Yaskawa INFORM job: OK_R2_O55A(90,180)KMOK.JBI

/JOB
//NAME OK_R2_O55A(90,180)KMOK
//POS
///NPOS 386,386,386,17,0,0
///TOOL 0
///POSTYPE PULSE
///PULSE
C00000=-76403,1922,-14330,-35191,82947,48006
C00001=-78901,2717,-11338,-34802,80748,47687
C00002=-84368,8537,-7735,-27600,82156,45752
C00003=-85611,7008,-9073,-27350,81787,45371
C00004=-84730,8997,-7223,-27533,81967,45660
C00005=-84730,9088,-5441,-27593,81032,45882
C00006=-85090,9461,-6706,-27466,81778,45569
C00007=-85585,11950,-4488,-27371,81540,45439
C00008=-80569,4182,-8968,-34529,79490,47402
C00009=-79583,3757,-10261,-34677,80367,47529
C00010=-77101,2900,-13311,-35064,82560,47846
C00011=-78635,-10836,-23571,-6788,56023,46567
C00012=-80100,-6638,-17370,-6019,54259,46080
C00013=-81067,-4347,-13182,-5518,52796,45761
C00014=-81067,-4111,-11404,-5589,51829,45816
C00015=-81465,-3918,-12726,-5271,52710,45599
C00016=-81982,-3205,-12144,-4945,52685,45384
C00017=-81465,-3918,-12726,-5271,52710,45599
C00018=-79282,-7726,-17487,-6563,53838,46443
C00019=-77787,-11932,-23670,-7341,55599,46936
C00020=-71781,-30779,-36927,-16583,56350,53193
C00021=-76601,7892,12119,-36699,72044,51538
C00022=-79081,9717,16128,-36650,69746,51261
C00023=-82756,10272,16118,-32252,68446,49901
C00024=-83910,8771,14784,-32035,68048,49533
C00025=-82756,10272,16118,-32252,68446,49901
C00026=-82756,11092,18536,-32472,67538,50179
C00027=-82756,10272,16118,-32252,68446,49901
C00028=-83393,13264,18808,-32164,68102,49736
C00029=-82756,10272,16118,-32252,68446,49901
C00030=-79125,8186,14884,-36648,69710,51254
C00031=-76625,6364,10892,-36701,72010,51539
C00032=-78619,-8468,-7802,-7622,47602,47178
C00033=-80084,-3545,-911,-6819,45772,46643
C00034=-80849,-1134,3864,-6473,44020,46410
C00035=-80849,-591,5622,-6568,43222,46468
C00036=-80849,-1134,3864,-6473,44020,46410
C00037=-81794,988,5635,-5793,43949,45962
C00038=-80849,-1134,3864,-6473,44020,46410
C00039=-79264,-4301,-246,-7489,45053,47087
C00040=-77768,-9252,-7148,-8299,46887,47630
C00041=-73501,-22878,-17280,-17361,48294,53822
C00042=-76582,7918,12198,-36708,72023,51553
C00043=-79062,9745,16210,-36660,69725,51276
C00044=-85631,8937,11684,-26093,69417,48444
C00045=-86788,7574,10485,-25849,69089,48061
C00046=-85631,8937,11684,-26093,69417,48444
C00047=-85631,9727,14257,-26282,68355,48694
C00048=-85631,8937,11684,-26093,69417,48444
C00049=-86384,12817,15152,-25960,69054,48229
C00050=-80206,9359,17079,-36653,68644,51156
C00051=-79213,8529,15380,-36663,69568,51266
C00052=-76716,6688,11367,-36712,71869,51549
C00053=-78496,-8401,-7547,-7720,47491,47244
C00054=-79964,-3473,-648,-6917,45658,46708
C00055=-80829,339,5196,-6494,43959,46423
C00056=-80829,927,7090,-6597,43101,46485
C00057=-80829,339,5196,-6494,43959,46423
C00058=-81723,1584,6242,-5853,43887,45997
C00059=-80829,339,5196,-6494,43959,46423
C00060=-79396,-4326,-472,-7381,45166,47015
C00061=-77904,-9273,-7368,-8190,46997,47557
C00062=-73798,-22065,-16698,-17164,48289,53685
C00063=-76687,8147,12453,-36701,71947,51534
C00064=-79164,9987,16479,-36654,69648,51259
C00065=-85469,9101,11403,-25682,69642,48313
C00066=-87077,7212,9743,-25336,69193,47776
C00067=-85469,9101,11403,-25682,69642,48313
C00068=-85469,10017,14410,-25899,68394,48603
C00069=-85469,9101,11403,-25682,69642,48313
C00070=-86200,12844,14752,-25552,69292,48104
C00071=-80097,9169,16882,-36663,68709,51181
C00072=-79103,8344,15188,-36673,69634,51291
C00073=-76603,6515,11188,-36723,71934,51575
C00074=-78620,-8311,-7590,-7627,47551,47182
C00075=-80084,-3383,-689,-6825,45719,46647
C00076=-80782,-115,4996,-6540,43852,46454
C00077=-80782,405,6668,-6631,43097,46512
C00078=-80782,126,5782,-6582,43497,46482
C00079=-81646,1735,7133,-5954,43425,46068
C00080=-80263,-769,3748,-6862,44325,46668
C00081=-79285,-4364,-387,-7468,45105,47073
C00082=-77789,-9311,-7283,-8278,46937,47615
C00083=-72207,-27183,-21377,-18066,48871,54317
C00084=-76718,8235,12740,-36721,71828,51562
C00085=-79194,10089,16780,-36678,69527,51288
C00086=-85949,10651,13260,-25494,69998,48201
C00087=-87185,9191,11962,-25242,69663,47789
C00088=-85949,10651,13260,-25494,69998,48201
C00089=-85949,11213,15096,-25622,69235,48375
C00090=-85949,10898,14078,-25551,69656,48279
C00091=-86536,13982,16861,-25455,69360,48114
C00092=-80117,8915,16512,-36639,68779,51146
C00093=-79122,8093,14823,-36651,69703,51257
C00094=-76620,6271,10832,-36704,72003,51543
C00095=-78696,-8281,-7580,-7575,47554,47147
C00096=-80158,-3350,-677,-6772,45721,46612
C00097=-80887,125,5361,-6477,43742,46411
C00098=-80887,585,6834,-6555,43076,46460
C00099=-80887,270,5831,-6501,43529,46426
C00100=-81591,1736,7061,-5991,43471,46090
C00101=-79799,-2298,2499,-7195,44348,46889
C00102=-79220,-4347,-358,-7515,45102,47104
C00103=-77723,-9293,-7254,-8324,46936,47646
C00104=-72435,-26599,-20972,-17915,48869,54211
C00105=-76570,-17687,-14850,-19798,75838,26477
C00106=-76570,-17687,-14850,-19798,75838,26477
C00107=-87745,-9605,-5375,-17930,71662,23017
C00108=-89443,-6815,-2798,-17604,71148,22465
C00109=-89634,-5842,-2020,-17563,71128,22397
C00110=-89443,-6815,-2798,-17604,71148,22465
C00111=-89443,-7581,-5630,-17479,72437,22273
C00112=-91168,1721,1990,-17114,72156,21677
C00113=-91168,2041,3217,-17166,71590,21758
C00114=-91168,1721,1990,-17114,72156,21677
C00115=-82202,21106,36308,-50868,81053,24298
C00116=-83204,19644,34921,-50948,80572,24044
C00117=-78958,6455,21071,-50417,84024,24348
C00118=-86052,-24055,-21651,-18038,74505,23209
C00119=-69214,24096,20749,-23108,83460,36221
C00120=-71608,6597,4603,-68947,81663,-45930
C00121=-73755,7964,8737,-69115,79508,-45414
C00122=-74968,7560,10682,-69317,78154,-44963
C00123=-74968,8346,13234,-69526,77715,-44454
C00124=-74968,7560,10682,-69317,78154,-44963
C00125=-75623,8350,11378,-69309,77705,-45039
C00126=-73234,7979,11391,-69373,79243,-44640
C00127=-72371,7345,9649,-69271,80108,-44853
C00128=-70208,5990,5521,-69090,82272,-45369
C00129=-71458,6536,4837,-68973,81696,-45835
C00130=-73608,7910,8978,-69146,79540,-45319
C00131=-74773,7989,11985,-69422,78068,-44683
C00132=-74773,8525,13689,-69560,77778,-44345
C00133=-74773,8199,12662,-69476,77952,-44548
C00134=-75530,9339,13667,-69477,77429,-44630
C00135=-73160,8336,11414,-69348,79357,-44704
C00136=-72299,7709,9679,-69249,80221,-44917
C00137=-70142,6374,5567,-69075,82381,-45433
C00138=-71555,6569,4727,-68960,81663,-45884
C00139=-73704,8675,11428,-69316,79052,-44847
C00140=-74869,8697,12280,-69388,78072,-44775
C00141=-74869,9238,14009,-69531,77776,-44434
C00142=-74869,8887,12896,-69439,77966,-44653
C00143=-75513,9557,13488,-69438,77523,-44728
C00144=-73243,7935,11201,-69359,79273,-44682
C00145=-72380,7304,9463,-69258,80138,-44894
C00146=-70217,5958,5343,-69080,82301,-45410
C00147=-71620,7576,9372,-69242,80725,-44881
C00148=-73772,8435,11320,-69324,78986,-44831
C00149=-74875,8509,12078,-69384,78077,-44787
C00150=-74875,9056,13841,-69527,77773,-44437
C00151=-74875,8686,12655,-69431,77977,-44672
C00152=-75602,9232,13138,-69428,77479,-44758
C00153=-73284,7952,11199,-69357,79249,-44692
C00154=-72421,7320,9461,-69256,80114,-44904
C00155=-70258,5972,5339,-69078,82277,-45419
C00156=-71548,6406,4570,-68959,81673,-45889
C00157=-73698,8629,11672,-69344,78990,-44771
C00158=-74886,8172,11775,-69381,78074,-44795
C00159=-74886,8662,13358,-69511,77801,-44479
C00160=-74886,8307,12218,-69417,77997,-44706
C00161=-75624,9078,12897,-69416,77490,-44791
C00162=-73253,7959,11238,-69360,79262,-44679
C00163=-72390,7327,9499,-69259,80127,-44891
C00164=-70227,5979,5377,-69081,82290,-45407
C00165=-73684,21924,28477,-69535,76234,-41822
C00166=-74891,19654,26327,-69526,75480,-42047
C00167=-76506,21387,29456,-69805,74005,-41798
C00168=-74552,18110,24880,-69499,75745,-42046
C00169=-75381,18098,23573,-69331,75487,-42506
C00170=-77346,18837,26951,-69763,73526,-42008
C00171=-78427,17842,26055,-69366,71469,-52011
C00172=-78881,15304,23707,-69325,71217,-52134
C00173=-74815,19796,26463,-68977,79664,-56247
C00174=-73178,22919,29433,-68939,80676,-55936
C00175=-73666,19272,20464,-68833,77604,-43382
C00176=-74869,18380,22636,-69174,76106,-42756
C00177=-76554,20444,27119,-69566,74331,-42226
C00178=-74527,17435,22965,-69319,76074,-42409
C00179=-75357,17458,21697,-69150,75817,-42866
C00180=-76969,16913,23840,-69520,74127,-42370
C00181=-77511,13158,20364,-69473,73839,-42534
C00182=-77277,24403,30938,-69278,81382,-40713
C00183=-74792,18886,23871,-68814,80114,-56732
C00184=-73159,20683,22818,-68588,81821,-57193
C00185=-73710,21944,28497,-69536,76216,-41825
C00186=-74917,19676,26348,-69527,75461,-42050
C00187=-76528,21588,29866,-69843,73933,-41733
C00188=-74578,18131,24900,-69499,75726,-42049
C00189=-75407,18120,23593,-69332,75469,-42509
C00190=-76893,18416,26783,-69784,73785,-41898
C00191=-77360,15711,24383,-69770,73503,-41999
C00192=-77117,25124,33254,-69494,80031,-40440
C00193=-77229,28421,36396,-69270,82410,-39863
C00194=-74841,19817,26484,-68979,79646,-56250
C00195=-73204,22940,29453,-68940,80658,-55939
C00196=-73671,21913,28467,-69535,76243,-41821
C00197=-74878,19644,26317,-69525,75489,-42046
C00198=-76446,21696,29741,-69776,74042,-41781
C00199=-74539,18100,24870,-69498,75754,-42045
C00200=-75368,18087,23562,-69331,75496,-42505
C00201=-76829,18736,26940,-69733,73861,-41920
C00202=-77356,15298,23767,-69695,73575,-42071
C00203=-77179,22049,30100,-69528,78702,-40871
C00204=-77429,20567,28688,-69524,78574,-40949
C00205=-74802,19785,26453,-68977,79673,-56246
C00206=-73165,22909,29423,-68938,80686,-55935
C00207=-73697,21934,28487,-69536,76225,-41823
C00208=-74904,19665,26338,-69526,75471,-42049
C00209=-76487,21502,29779,-69838,73968,-41730
C00210=-74565,18121,24890,-69499,75735,-42048
C00211=-75394,18109,23583,-69331,75478,-42508
C00212=-76921,18139,26617,-69792,73759,-41884
C00213=-77416,14929,23641,-69755,73493,-42028
C00214=-76976,35689,43864,-68952,85010,-38929
C00215=-77187,33996,42040,-68958,84967,-39065
C00216=-74828,19807,26473,-68978,79655,-56248
C00217=-71271,31949,38327,-68936,81632,-55329
C00218=-64455,21408,16051,-68515,88030,-41500
C00219=-62220,-14655,-7588,-61843,66390,-57480
C00220=-65684,-34059,-16244,-44657,38104,-81353
C00221=-80507,10121,17600,-15341,57200,39800
C00222=-75845,16867,22558,-16973,58521,41505
C00223=-72897,41582,49979,-26317,62594,52964
C00224=-79860,8562,16225,-15575,57367,40041
C00225=-80508,9482,15745,-15208,57986,39686
C00226=-72982,41184,49489,-26278,62657,52914
C00227=-73697,37517,45702,-26032,62835,52576
C00228=-77058,24794,32654,-21193,59755,46647
C00229=-81408,13297,22074,-15190,55949,39611
C00230=-82232,11238,20195,-14857,55894,39277
C00231=-83257,9100,18238,-14442,55814,38864
C00232=-84450,6933,16333,-13966,55662,38392
C00233=-78697,11090,18471,-9995,55076,34572
C00234=-79295,11807,19109,-9744,54979,34335
C00235=-80544,10273,17728,-36477,70612,65921
C00236=-80540,10255,17715,-36477,70612,65923
C00237=-81663,12108,20960,-36551,69289,65897
C00238=-80539,9618,15857,-36320,71277,65692
C00239=-79786,11468,18802,-36578,70896,66153
C00240=-81901,13148,21842,-36522,69179,65831
C00241=-83549,20571,28688,-36398,68155,65466
C00242=-80537,10245,17705,-38455,66333,65488
C00243=-80540,10262,17718,-38454,66333,65487
C00244=-77732,-5014,-1669,-37983,70842,65115
C00245=-70423,-28857,-26484,-34936,42937,-87209
C00246=-72957,-20656,-20669,-25335,39181,70937
C00247=-76432,-9207,-9095,-22895,37031,69584
C00248=-77636,-3976,-2319,-22541,35326,69388
C00249=-76934,-7535,-7865,-22379,36987,69297
C00250=-76131,-8379,-7270,-23539,36472,69943
C00251=-76886,-1544,-324,-23246,35556,69779
C00252=-76079,1584,2343,-24028,35756,70214
C00253=-76929,-7527,-7764,-26477,38278,71586
C00254=-75666,-12476,-14553,-26648,40152,71669
C00255=-80539,4002,-16743,-13402,74658,37601
C00256=-80536,3873,-13936,-13516,72912,37797
C00257=-81546,5662,-9698,-13281,71105,37640
C00258=-79886,2359,-14058,-13789,72336,38095
C00259=-80534,3865,-14021,-13513,72959,37793
C00260=-82537,3680,-11348,-12920,70949,37307
C00261=-83585,1661,-13067,-12546,70807,36945
C00262=-84541,-32,-14546,-12201,70702,36611
C00263=-79182,4632,-13287,-8514,71050,33082
C00264=-78761,4323,-16471,-8590,72875,33101
C00265=-80569,4030,-12503,-34597,83280,61769
C00266=-80562,4114,-9678,-34698,81876,62211
C00267=-81659,4236,-6801,-34632,80014,62350
C00268=-80559,4091,-9841,-34693,81950,62189
C00269=-79806,5370,-7496,-34879,81603,62605
C00270=-82051,6116,-5182,-34562,79830,62247
C00271=-83492,12161,48,-34308,79156,61868
C00272=-83703,13184,961,-34271,79043,61817
C00273=-80556,4261,-7630,-36043,76415,61879
C00274=-80562,4081,-10441,-35844,77751,61431
C00275=-71462,-12551,-24032,-37751,81493,64028
C00276=-64215,-41183,-30200,-41548,42479,-83127
C00277=-75268,-8940,1587,-28059,31543,72401
C00278=-76569,-4731,4953,-26676,31199,71625
C00279=-77625,506,10820,-26265,30038,71368
C00280=-77071,-3623,4563,-25583,31771,71034
C00281=-76271,-4245,5350,-26977,31300,71794
C00282=-76971,2980,13032,-27029,30166,71792
C00283=-76158,6294,15992,-27966,30325,72317
C00284=-77064,-3050,6321,-30619,32600,73861
C00285=-75803,-7249,2926,-31827,33007,74555
C00286=-80516,10172,17645,-15338,57197,39797
C00287=-80517,10165,17644,-15338,57194,39797
C00288=-81429,13162,21998,-15186,55919,39607
C00289=-79869,8613,16269,-15572,57363,40038
C00290=-80517,9533,15790,-15205,57982,39683
C00291=-82245,11269,20291,-14856,55845,39281
C00292=-83580,8472,17804,-14322,55699,38749
C00293=-84398,6972,16513,-13999,55581,38427
C00294=-79088,10454,17905,-9826,55051,34413
C00295=-74888,4098,12338,-11562,55761,36069
C00296=-80552,10324,17774,-36476,70606,65919
C00297=-80549,10306,17761,-36476,70607,65921
C00298=-83683,7693,15438,-32682,67636,65344
C00299=-80548,9669,15902,-36319,71272,65690
C00300=-79795,11519,18847,-36577,70890,66151
C00301=-84004,9174,16701,-32630,67499,65250
C00302=-85602,16570,23210,-32388,66714,64811
C00303=-80546,10295,17751,-38454,66328,65486
C00304=-80549,10312,17763,-38453,66327,65485
C00305=-76939,-6698,-208,-38485,69790,65864
C00306=-67266,-29602,-13484,-36434,33447,77204
C00307=-75146,-9337,1276,-28189,31574,72475
C00308=-76453,-5135,4625,-26799,31231,71694
C00309=-77647,460,10904,-26298,29964,71381
C00310=-76958,-4030,4231,-25703,31802,71100
C00311=-76155,-4648,5022,-27099,31332,71863
C00312=-76931,2821,12923,-27078,30166,71815
C00313=-76073,5866,15538,-28006,30408,72336
C00314=-76950,-3457,5988,-30727,32638,73923
C00315=-75683,-7648,2608,-31942,33044,74622
C00316=-80508,8315,12089,-14954,59582,39461
C00317=-80505,9651,16284,-15248,57749,39721
C00318=-81490,12944,21701,-15149,55979,39575
C00319=-79855,8537,16203,-15577,57368,40043
C00320=-80504,9457,15722,-15209,57987,39688
C00321=-82467,11028,20074,-14770,55816,39193
C00322=-83319,9325,18634,-14437,55675,38860
C00323=-83964,7971,17403,-14174,55621,38599
C00324=-84422,7198,16724,-13991,55562,38417
C00325=-78819,10126,16706,-9875,55645,34468
C00326=-78596,10216,16456,-9945,55869,34539
C00327=-80539,10247,17706,-36477,70615,65922
C00328=-80536,10230,17693,-36477,70615,65924
C00329=-81604,11432,20382,-36558,69320,65911
C00330=-80534,9593,15834,-36320,71280,65693
C00331=-79781,11443,18779,-36578,70899,66154
C00332=-82039,13393,22124,-36517,69083,65803
C00333=-83392,19347,27632,-36414,68242,65504
C00334=-83616,20496,28669,-36395,68109,65452
C00335=-80533,10219,17683,-38456,66335,65489
C00336=-80536,10236,17695,-38455,66335,65488
C00337=-76398,-4716,5168,-39090,68227,66710
C00338=-67688,-28685,-12865,-36008,33343,76954
C00339=-75228,-9072,1484,-28102,31553,72426
C00340=-76531,-4865,4844,-26717,31210,71648
C00341=-77847,119,10662,-26106,29876,71275
C00342=-77033,-3758,4453,-25623,31782,71056
C00343=-76233,-4379,5241,-27017,31310,71817
C00344=-76936,2995,13152,-27116,30117,71837
C00345=-76130,6238,16052,-28051,30278,72358
C00346=-77026,-3185,6210,-30655,32612,73882
C00347=-75763,-7381,2820,-31865,33019,74577
C00348=-80512,10146,17623,-15339,57198,39799
C00349=-80513,10140,17621,-15339,57196,39799
C00350=-81500,13127,22067,-15170,55850,39589
C00351=-79864,8588,16247,-15574,57365,40040
C00352=-80513,9508,15768,-15206,57984,39684
C00353=-82364,10966,20070,-14819,55805,39239
C00354=-83277,9255,18611,-14462,55660,38880
C00355=-83996,7868,17423,-14178,55551,38597
C00356=-84389,7230,16943,-14028,55450,38448
C00357=-78699,12714,19934,-10002,55011,34578
C00358=-77475,15494,24062,-10661,54073,35179
C00359=-80548,10298,17751,-36476,70609,65920
C00360=-80545,10281,17738,-36477,70610,65922
C00361=-82679,9625,18013,-34629,68410,65635
C00362=-80543,9644,15879,-36319,71274,65691
C00363=-79790,11494,18824,-36577,70893,66152
C00364=-83022,11356,19462,-34579,68269,65534
C00365=-84222,16885,24482,-34449,67579,65242
C00366=-84495,18260,25693,-34414,67437,65171
C00367=-80541,10270,17728,-38455,66331,65487
C00368=-80544,10287,17740,-38454,66331,65486
C00369=-71600,-1949,10031,-39049,69350,68326
C00370=-71600,-1949,10031,-39049,69350,68326
C00371=-78766,16664,26924,-37375,68202,69313
C00372=-80481,18381,29464,-37332,66914,69021
C00373=-80571,20050,31036,-37349,66789,69027
C00374=-82589,28813,39248,-37227,65478,68604
C00375=-78367,25278,33930,-37393,68464,69394
C00376=-93563,26241,26451,4282,61542,63605
C00377=-96314,32508,36024,18641,58909,62055
C00378=-92113,24530,27996,5482,55270,70397
C00379=-92106,24462,27769,4672,55649,70406
C00380=-91576,23902,26334,-3618,58754,70962
C00381=-93650,12043,18084,-5384,52096,70498
C00382=-97507,8799,15190,-3438,51997,68869
C00383=-93212,4360,14554,-16260,47827,71925
C00384=-94425,-6257,-911,-4852,54321,70064
C00385=-44833,-55261,-28957,-41445,79036,76616
BC00000=349204,673109,1075175
BC00001=349204,673109,1075175
BC00002=349204,673109,1075175
BC00003=349204,673109,1075175
BC00004=349204,673109,1075175
BC00005=349204,673109,1075175
BC00006=349204,673109,1075175
BC00007=349204,673109,1075175
BC00008=349204,673109,1075175
BC00009=349204,673109,1075175
BC00010=349204,673109,1075175
BC00011=305088,674616,1075175
BC00012=305088,674616,1075175
BC00013=305088,674616,1075175
BC00014=305088,674616,1075175
BC00015=305088,674616,1075175
BC00016=305088,674616,1075175
BC00017=305088,674616,1075175
BC00018=305088,674616,1075175
BC00019=305088,674616,1075175
BC00020=314803,666681,1075175
BC00021=348681,674864,1042481
BC00022=348681,674864,1042481
BC00023=348681,674864,1042481
BC00024=348681,674864,1042481
BC00025=348681,674864,1042481
BC00026=348681,674864,1042481
BC00027=348681,674864,1042481
BC00028=348681,674864,1042481
BC00029=348681,674864,1042481
BC00030=348681,674864,1042481
BC00031=348681,674864,1042481
BC00032=304891,674718,1003525
BC00033=304891,674718,1003525
BC00034=304891,674718,1003525
BC00035=304891,674718,1003525
BC00036=304891,674718,1003525
BC00037=304891,674718,1003525
BC00038=304891,674718,1003525
BC00039=304891,674718,1003525
BC00040=304891,674718,1003525
BC00041=314838,666681,1004817
BC00042=348633,674683,878796
BC00043=348633,674683,878796
BC00044=348633,674683,878796
BC00045=348633,674683,878796
BC00046=348633,674683,878796
BC00047=348633,674683,878796
BC00048=348633,674683,878796
BC00049=348633,674683,878796
BC00050=348633,674683,878796
BC00051=348633,674683,878796
BC00052=348633,674683,878796
BC00053=305592,674868,842714
BC00054=305592,674868,842714
BC00055=305592,674868,842714
BC00056=305592,674868,842714
BC00057=305592,674868,842714
BC00058=305592,674868,842714
BC00059=305592,674868,842714
BC00060=305592,674868,842714
BC00061=305592,674868,842714
BC00062=314872,666681,843515
BC00063=348685,675197,716542
BC00064=348685,675197,716542
BC00065=348685,675197,716542
BC00066=348685,675197,716542
BC00067=348685,675197,716542
BC00068=348685,675197,716542
BC00069=348685,675197,716542
BC00070=348685,675197,716542
BC00071=348685,675197,716542
BC00072=348685,675197,716542
BC00073=348685,675197,716542
BC00074=305467,675287,679878
BC00075=305467,675287,679878
BC00076=305467,675287,679878
BC00077=305467,675287,679878
BC00078=305467,675287,679878
BC00079=305467,675287,679878
BC00080=305467,675287,679878
BC00081=305467,675287,679878
BC00082=305467,675287,679878
BC00083=314907,666681,682214
BC00084=348720,675488,554835
BC00085=348720,675488,554835
BC00086=348720,675488,554835
BC00087=348720,675488,554835
BC00088=348720,675488,554835
BC00089=348720,675488,554835
BC00090=348720,675488,554835
BC00091=348720,675488,554835
BC00092=348720,675488,554835
BC00093=348720,675488,554835
BC00094=348720,675488,554835
BC00095=305310,675530,518487
BC00096=305310,675530,518487
BC00097=305310,675530,518487
BC00098=305310,675530,518487
BC00099=305310,675530,518487
BC00100=305310,675530,518487
BC00101=305310,675530,518487
BC00102=305310,675530,518487
BC00103=305310,675530,518487
BC00104=314942,666681,520912
BC00105=378648,679076,578921
BC00106=378648,679076,319795
BC00107=378648,679076,319795
BC00108=378648,679076,319795
BC00109=378648,679076,319795
BC00110=378648,679076,319795
BC00111=378648,679076,319795
BC00112=378648,679076,319795
BC00113=378648,679076,319795
BC00114=378648,679076,319795
BC00115=378648,679076,319795
BC00116=378648,679076,319795
BC00117=378648,679076,319795
BC00118=378648,679076,319795
BC00119=378648,679076,578921
BC00120=398174,688559,405806
BC00121=398174,688559,405806
BC00122=398174,688559,405806
BC00123=398174,688559,405806
BC00124=398174,688559,405806
BC00125=398174,688559,405806
BC00126=398174,688559,405806
BC00127=398174,688559,405806
BC00128=398174,688559,405806
BC00129=398174,688393,568935
BC00130=398174,688393,568935
BC00131=398174,688393,568935
BC00132=398174,688393,568935
BC00133=398174,688393,568935
BC00134=398174,688393,568935
BC00135=398174,688393,568935
BC00136=398174,688393,568935
BC00137=398174,688393,568935
BC00138=398174,688149,730160
BC00139=398174,688149,730160
BC00140=398174,688149,730160
BC00141=398174,688149,730160
BC00142=398174,688149,730160
BC00143=398174,688149,730160
BC00144=398174,688149,730160
BC00145=398174,688149,730160
BC00146=398174,688149,730160
BC00147=398174,687828,892370
BC00148=398174,687828,892370
BC00149=398174,687828,892370
BC00150=398174,687828,892370
BC00151=398174,687828,892370
BC00152=398174,687828,892370
BC00153=398174,687828,892370
BC00154=398174,687828,892370
BC00155=398174,687828,892370
BC00156=398174,687735,1053470
BC00157=398174,687735,1053470
BC00158=398174,687735,1053470
BC00159=398174,687735,1053470
BC00160=398174,687735,1053470
BC00161=398174,687735,1053470
BC00162=398174,687735,1053470
BC00163=398174,687735,1053470
BC00164=398174,687735,1053470
BC00165=398174,675730,786203
BC00166=398174,679514,767318
BC00167=398174,681028,759764
BC00168=398174,681028,759764
BC00169=398174,681028,759764
BC00170=398174,679196,759749
BC00171=398174,676312,759427
BC00172=398174,676312,759427
BC00173=398174,682565,762575
BC00174=398174,680140,779769
BC00175=398174,675445,1075175
BC00176=398174,679229,1075175
BC00177=398174,680743,1075175
BC00178=398174,680743,1075175
BC00179=398174,680743,1075175
BC00180=398174,680743,1075175
BC00181=398174,680743,1075175
BC00182=398174,680743,1075175
BC00183=398174,682279,1075175
BC00184=398174,679854,1075175
BC00185=398174,676016,462794
BC00186=398174,679800,443908
BC00187=398174,681314,436354
BC00188=398174,681314,436354
BC00189=398174,681314,436354
BC00190=398174,681314,436354
BC00191=398174,681314,436354
BC00192=398174,681314,436354
BC00193=398174,681314,436354
BC00194=398174,682851,439165
BC00195=398174,680426,456359
BC00196=398174,675587,948311
BC00197=398174,679371,929426
BC00198=398174,680885,921868
BC00199=398174,680885,921872
BC00200=398174,680885,921872
BC00201=398174,680885,921868
BC00202=398174,680885,921868
BC00203=398174,680885,921868
BC00204=398174,680885,921868
BC00205=398174,682422,924682
BC00206=398174,679997,941876
BC00207=398174,675874,624095
BC00208=398174,679658,605210
BC00209=398174,681170,597651
BC00210=398174,681171,597656
BC00211=398174,681171,597656
BC00212=398174,681170,597651
BC00213=398174,681170,597651
BC00214=398174,681170,597651
BC00215=398174,681170,597651
BC00216=398174,682708,600466
BC00217=398174,680283,617660
BC00218=398174,666681,626567
BC00219=360198,666681,720930
BC00220=313360,666681,837312
BC00221=317534,668949,937568
BC00222=315368,674001,918688
BC00223=314501,676022,911136
BC00224=314501,676022,911136
BC00225=314501,676022,911136
BC00226=314501,676022,911136
BC00227=314501,676022,911136
BC00228=314501,676022,911136
BC00229=314501,676022,911136
BC00230=314501,676022,911136
BC00231=314501,676022,911136
BC00232=314501,676022,911136
BC00233=293205,672518,918719
BC00234=294306,667154,937598
BC00235=358411,669398,910199
BC00236=352988,671786,892375
BC00237=350819,672740,885243
BC00238=350819,672741,885245
BC00239=350819,672741,885245
BC00240=350819,672741,885245
BC00241=350819,672741,885245
BC00242=349387,669987,879930
BC00243=354654,666972,897113
BC00244=354755,666681,897949
BC00245=313290,666681,1075175
BC00246=299789,666220,1075175
BC00247=298966,666220,1075175
BC00248=298637,666220,1075175
BC00249=298637,666220,1075175
BC00250=298637,666220,1075175
BC00251=298637,666220,1075175
BC00252=298637,666220,1075175
BC00253=311807,666220,1075175
BC00254=312962,666220,1075175
BC00255=317588,668663,1075175
BC00256=315422,673716,1075175
BC00257=314555,675737,1075175
BC00258=314555,675737,1075175
BC00259=314555,675737,1075175
BC00260=314556,675736,1075175
BC00261=314556,675736,1075175
BC00262=314556,675736,1075175
BC00263=293260,672232,1075175
BC00264=294360,666869,1075175
BC00265=358465,669112,1075175
BC00266=353042,671500,1075175
BC00267=350873,672456,1075175
BC00268=350873,672456,1075175
BC00269=350873,672456,1075175
BC00270=350873,672456,1075175
BC00271=350873,672456,1075175
BC00272=350873,672456,1075175
BC00273=349450,669548,1075175
BC00274=354717,666534,1075175
BC00275=354685,666681,1075175
BC00276=313430,666681,513902
BC00277=299680,666220,513222
BC00278=298858,666220,494557
BC00279=298529,666220,487091
BC00280=298529,666220,487091
BC00281=298529,666220,487091
BC00282=298529,666220,487091
BC00283=298529,666220,487091
BC00284=311698,666220,494536
BC00285=312853,666220,513199
BC00286=317480,669234,614158
BC00287=315313,674287,595278
BC00288=314447,676308,587726
BC00289=314447,676308,587726
BC00290=314447,676308,587726
BC00291=314447,676308,587726
BC00292=314447,676308,587726
BC00293=314447,676308,587726
BC00294=293151,672804,595309
BC00295=294252,667440,614188
BC00296=358357,669683,586789
BC00297=352934,672071,568965
BC00298=350764,673027,561835
BC00299=350764,673027,561835
BC00300=350764,673027,561835
BC00301=350764,673027,561835
BC00302=350764,673027,561835
BC00303=349300,670887,556521
BC00304=354567,667872,573704
BC00305=354825,666681,574539
BC00306=299762,666220,998740
BC00307=299762,666220,998740
BC00308=298939,666220,980075
BC00309=298610,666220,972608
BC00310=298610,666220,972608
BC00311=298610,666220,972608
BC00312=298610,666220,972608
BC00313=298610,666220,972608
BC00314=311779,666220,980053
BC00315=312935,666220,998717
BC00316=317561,668805,1075175
BC00317=315395,673858,1075175
BC00318=314528,675879,1073244
BC00319=314528,675879,1073244
BC00320=314528,675879,1073244
BC00321=314528,675879,1073244
BC00322=314528,675879,1073244
BC00323=314528,675879,1073244
BC00324=314528,675879,1073244
BC00325=293232,672375,1075175
BC00326=294333,667011,1075175
BC00327=358439,669255,1072306
BC00328=353015,671643,1054482
BC00329=350846,672598,1047353
BC00330=350846,672598,1047353
BC00331=350846,672598,1047353
BC00332=350846,672598,1047353
BC00333=350846,672598,1047353
BC00334=350846,672598,1047353
BC00335=349348,671076,1042041
BC00336=354615,668061,1059224
BC00337=354720,666681,1060057
BC00338=299707,666220,674523
BC00339=299707,666220,674523
BC00340=298885,666220,655858
BC00341=298556,666220,648392
BC00342=298556,666220,648392
BC00343=298556,666220,648392
BC00344=298556,666220,648392
BC00345=298556,666220,648392
BC00346=311725,666220,655837
BC00347=312880,666220,674501
BC00348=317507,669092,775460
BC00349=315340,674145,756580
BC00350=314474,676166,749028
BC00351=314474,676166,749028
BC00352=314474,676166,749028
BC00353=314474,676166,749028
BC00354=314474,676166,749028
BC00355=314474,676166,749028
BC00356=314474,676166,749028
BC00357=293178,672661,756610
BC00358=294279,667297,775489
BC00359=358384,669541,748090
BC00360=352961,671929,730266
BC00361=350791,672884,723137
BC00362=350791,672884,723137
BC00363=350791,672884,723137
BC00364=350791,672884,723137
BC00365=350791,672884,723137
BC00366=350791,672884,723137
BC00367=349368,669977,717821
BC00368=354635,666962,735004
BC00369=354635,666962,735004
BC00370=343366,666962,351655
BC00371=343366,666962,351655
BC00372=343366,666962,351655
BC00373=343366,666962,351655
BC00374=343366,666962,351655
BC00375=343366,666962,351655
BC00376=343366,666962,351655
BC00377=343366,666962,351655
BC00378=343366,666962,351655
BC00379=343366,666962,351655
BC00380=343366,666962,351655
BC00381=343366,666962,351655
BC00382=343366,666962,351655
BC00383=343366,666962,351655
BC00384=343366,666962,351655
BC00385=354635,666962,735004
EC00000=798156,1112951
EC00001=798156,1112951
EC00002=798156,1112951
EC00003=798156,1112951
EC00004=798156,1112951
EC00005=798156,1112951
EC00006=798156,1112951
EC00007=798156,1112951
EC00008=798156,1112951
EC00009=798156,1112951
EC00010=798156,1112951
EC00011=798156,1112951
EC00012=798156,1112951
EC00013=798156,1112951
EC00014=798156,1112951
EC00015=798156,1112951
EC00016=798156,1112951
EC00017=798156,1112951
EC00018=798156,1112951
EC00019=798156,1112951
EC00020=798156,1112951
EC00021=798156,1112951
EC00022=798156,1112951
EC00023=798156,1112951
EC00024=798156,1112951
EC00025=798156,1112951
EC00026=798156,1112951
EC00027=798156,1112951
EC00028=798156,1112951
EC00029=798156,1112951
EC00030=798156,1112951
EC00031=798156,1112951
EC00032=798156,1112951
EC00033=798156,1112951
EC00034=798156,1112951
EC00035=798156,1112951
EC00036=798156,1112951
EC00037=798156,1112951
EC00038=798156,1112951
EC00039=798156,1112951
EC00040=798156,1112951
EC00041=798156,1112951
EC00042=798156,1112951
EC00043=798156,1112951
EC00044=798156,1112951
EC00045=798156,1112951
EC00046=798156,1112951
EC00047=798156,1112951
EC00048=798156,1112951
EC00049=798156,1112951
EC00050=798156,1112951
EC00051=798156,1112951
EC00052=798156,1112951
EC00053=798156,1112951
EC00054=798156,1112951
EC00055=798156,1112951
EC00056=798156,1112951
EC00057=798156,1112951
EC00058=798156,1112951
EC00059=798156,1112951
EC00060=798156,1112951
EC00061=798156,1112951
EC00062=798156,1112951
EC00063=798156,1112951
EC00064=798156,1112951
EC00065=798156,1112951
EC00066=798156,1112951
EC00067=798156,1112951
EC00068=798156,1112951
EC00069=798156,1112951
EC00070=798156,1112951
EC00071=798156,1112951
EC00072=798156,1112951
EC00073=798156,1112951
EC00074=798156,1112951
EC00075=798156,1112951
EC00076=798156,1112951
EC00077=798156,1112951
EC00078=798156,1112951
EC00079=798156,1112951
EC00080=798156,1112951
EC00081=798156,1112951
EC00082=798156,1112951
EC00083=798156,1112951
EC00084=798156,1112951
EC00085=798156,1112951
EC00086=798156,1112951
EC00087=798156,1112951
EC00088=798156,1112951
EC00089=798156,1112951
EC00090=798156,1112951
EC00091=798156,1112951
EC00092=798156,1112951
EC00093=798156,1112951
EC00094=798156,1112951
EC00095=798156,1112951
EC00096=798156,1112951
EC00097=798156,1112951
EC00098=798156,1112951
EC00099=798156,1112951
EC00100=798156,1112951
EC00101=798156,1112951
EC00102=798156,1112951
EC00103=798156,1112951
EC00104=798156,1112951
EC00105=798156,1112951
EC00106=798156,1112951
EC00107=798156,1112951
EC00108=798156,1112951
EC00109=798156,1112951
EC00110=798156,1112951
EC00111=798156,1112951
EC00112=798156,1112951
EC00113=798156,1112951
EC00114=798156,1112951
EC00115=798156,1112951
EC00116=798156,1112951
EC00117=798156,1112951
EC00118=798156,1112951
EC00119=798156,1112951
EC00120=798156,1112951
EC00121=798156,1112951
EC00122=798156,1112951
EC00123=798156,1112951
EC00124=798156,1112951
EC00125=798156,1112951
EC00126=798156,1112951
EC00127=798156,1112951
EC00128=798156,1112951
EC00129=798156,1112951
EC00130=798156,1112951
EC00131=798156,1112951
EC00132=798156,1112951
EC00133=798156,1112951
EC00134=798156,1112951
EC00135=798156,1112951
EC00136=798156,1112951
EC00137=798156,1112951
EC00138=798156,1112951
EC00139=798156,1112951
EC00140=798156,1112951
EC00141=798156,1112951
EC00142=798156,1112951
EC00143=798156,1112951
EC00144=798156,1112951
EC00145=798156,1112951
EC00146=798156,1112951
EC00147=798156,1112951
EC00148=798156,1112951
EC00149=798156,1112951
EC00150=798156,1112951
EC00151=798156,1112951
EC00152=798156,1112951
EC00153=798156,1112951
EC00154=798156,1112951
EC00155=798156,1112951
EC00156=798156,1112951
EC00157=798156,1112951
EC00158=798156,1112951
EC00159=798156,1112951
EC00160=798156,1112951
EC00161=798156,1112951
EC00162=798156,1112951
EC00163=798156,1112951
EC00164=798156,1112951
EC00165=798156,1112951
EC00166=798156,1112951
EC00167=798156,1112951
EC00168=798156,1112951
EC00169=798156,1112951
EC00170=798156,1112951
EC00171=798156,1112951
EC00172=798156,1112951
EC00173=798156,1112951
EC00174=798156,1112951
EC00175=798156,1112951
EC00176=798156,1112951
EC00177=798156,1112951
EC00178=798156,1112951
EC00179=798156,1112951
EC00180=798156,1112951
EC00181=798156,1112951
EC00182=798156,1112951
EC00183=798156,1112951
EC00184=798156,1112951
EC00185=798156,1112951
EC00186=798156,1112951
EC00187=798156,1112951
EC00188=798156,1112951
EC00189=798156,1112951
EC00190=798156,1112951
EC00191=798156,1112951
EC00192=798156,1112951
EC00193=798156,1112951
EC00194=798156,1112951
EC00195=798156,1112951
EC00196=798156,1112951
EC00197=798156,1112951
EC00198=798152,1112950
EC00199=798156,1112951
EC00200=798156,1112951
EC00201=798152,1112950
EC00202=798152,1112950
EC00203=798152,1112950
EC00204=798152,1112950
EC00205=798156,1112951
EC00206=798156,1112951
EC00207=798156,1112951
EC00208=798156,1112951
EC00209=798153,1112948
EC00210=798156,1112951
EC00211=798156,1112951
EC00212=798153,1112948
EC00213=798153,1112948
EC00214=798153,1112948
EC00215=798153,1112948
EC00216=798156,1112951
EC00217=798156,1112951
EC00218=798156,1112951
EC00219=798156,1112951
EC00220=798156,1112951
EC00221=798156,1112951
EC00222=798156,1112951
EC00223=798156,1112951
EC00224=798156,1112951
EC00225=798156,1112951
EC00226=798156,1112951
EC00227=798156,1112951
EC00228=798156,1112951
EC00229=798156,1112951
EC00230=798156,1112951
EC00231=798156,1112951
EC00232=798156,1112951
EC00233=798156,1112951
EC00234=798156,1112951
EC00235=798156,1112951
EC00236=798156,1112951
EC00237=798154,1112950
EC00238=798156,1112951
EC00239=798156,1112951
EC00240=798156,1112951
EC00241=798156,1112951
EC00242=798156,1112951
EC00243=798156,1112951
EC00244=798156,1112951
EC00245=798156,1112951
EC00246=798156,1112951
EC00247=798156,1112951
EC00248=798156,1112951
EC00249=798156,1112951
EC00250=798156,1112951
EC00251=798156,1112951
EC00252=798156,1112951
EC00253=798156,1112951
EC00254=798156,1112951
EC00255=798156,1112951
EC00256=798156,1112951
EC00257=798156,1112951
EC00258=798156,1112951
EC00259=798156,1112951
EC00260=798155,1112950
EC00261=798155,1112950
EC00262=798155,1112950
EC00263=798156,1112951
EC00264=798156,1112951
EC00265=798156,1112951
EC00266=798156,1112951
EC00267=798156,1112951
EC00268=798156,1112951
EC00269=798156,1112951
EC00270=798156,1112951
EC00271=798156,1112951
EC00272=798156,1112951
EC00273=798156,1112951
EC00274=798156,1112951
EC00275=798156,1112951
EC00276=798156,1112951
EC00277=798156,1112951
EC00278=798156,1112951
EC00279=798156,1112951
EC00280=798156,1112951
EC00281=798156,1112951
EC00282=798156,1112951
EC00283=798156,1112951
EC00284=798156,1112951
EC00285=798156,1112951
EC00286=798156,1112951
EC00287=798156,1112951
EC00288=798156,1112951
EC00289=798156,1112951
EC00290=798156,1112951
EC00291=798156,1112951
EC00292=798156,1112951
EC00293=798156,1112951
EC00294=798156,1112951
EC00295=798156,1112951
EC00296=798156,1112951
EC00297=798156,1112951
EC00298=798156,1112951
EC00299=798156,1112951
EC00300=798156,1112951
EC00301=798156,1112951
EC00302=798156,1112951
EC00303=798156,1112951
EC00304=798156,1112951
EC00305=798156,1112951
EC00306=798156,1112951
EC00307=798156,1112951
EC00308=798156,1112951
EC00309=798156,1112951
EC00310=798156,1112951
EC00311=798156,1112951
EC00312=798156,1112951
EC00313=798156,1112951
EC00314=798156,1112951
EC00315=798156,1112951
EC00316=798156,1112951
EC00317=798156,1112951
EC00318=798156,1112951
EC00319=798156,1112951
EC00320=798156,1112951
EC00321=798156,1112951
EC00322=798156,1112951
EC00323=798156,1112951
EC00324=798156,1112951
EC00325=798156,1112951
EC00326=798156,1112951
EC00327=798156,1112951
EC00328=798156,1112951
EC00329=798156,1112951
EC00330=798156,1112951
EC00331=798156,1112951
EC00332=798156,1112951
EC00333=798156,1112951
EC00334=798156,1112951
EC00335=798156,1112951
EC00336=798156,1112951
EC00337=798156,1112951
EC00338=798156,1112951
EC00339=798156,1112951
EC00340=798156,1112951
EC00341=798156,1112951
EC00342=798156,1112951
EC00343=798156,1112951
EC00344=798156,1112951
EC00345=798156,1112951
EC00346=798156,1112951
EC00347=798156,1112951
EC00348=798156,1112951
EC00349=798156,1112951
EC00350=798156,1112951
EC00351=798156,1112951
EC00352=798156,1112951
EC00353=798156,1112951
EC00354=798156,1112951
EC00355=798156,1112951
EC00356=798156,1112951
EC00357=798156,1112951
EC00358=798156,1112951
EC00359=798156,1112951
EC00360=798156,1112951
EC00361=798156,1112951
EC00362=798156,1112951
EC00363=798156,1112951
EC00364=798156,1112951
EC00365=798156,1112951
EC00366=798156,1112951
EC00367=798156,1112951
EC00368=798156,1112951
EC00369=798156,1112951
EC00370=798156,1112951
EC00371=798156,1112951
EC00372=798156,1112951
EC00373=798156,1112951
EC00374=798156,1112951
EC00375=798156,1112951
EC00376=798156,1112951
EC00377=798156,1112951
EC00378=798156,1112951
EC00379=798156,1112951
EC00380=798156,1112951
EC00381=798156,1112951
EC00382=798156,1112951
EC00383=798156,1112951
EC00384=798156,1112951
EC00385=798156,1112951
///POSTYPE BASE
///RECTAN
///RCONF 0,0,0,0,0,0,0,0,0,0,0,0,0,0,0,0,0,0,0,0,0,0,0,0
P00006=0.222,-3.123,-1.508,0.0000,0.0000,0.0000
P00021=-0.225,-6.128,-0.405,0.0000,0.0000,0.0000
P00022=0.222,-3.123,-1.508,0.0000,0.0000,0.0000
P00023=0.143,-0.036,0.682,0.0000,0.0000,0.0000
P00031=1.853,-0.001,-1.549,0.0000,0.0000,0.0000
P00032=1.957,0.503,-7.217,0.0000,0.0000,0.0000
///RCONF 0,0,0,0,1,0,0,0,0,0,0,0,0,0,0,0,0,0,0,0,0,0,0,0
P00033=-0.123,0.612,-5.012,0.0000,0.0000,0.0000
///RCONF 0,0,0,0,0,0,0,0,0,0,0,0,0,0,0,0,0,0,0,0,0,0,0,0
P00041=0.192,3.924,0.305,0.0000,0.0000,0.0000
P00042=-0.217,1.941,0.413,0.0000,0.0000,0.0000
P00043=-0.044,-1.937,1.197,0.0000,0.0000,0.0000
P00051=0.367,3.892,0.009,0.0000,0.0000,0.0000
P00052=0.088,2.832,-0.342,0.0000,0.0000,0.0000
P00053=0.134,6.594,0.107,0.0000,0.0000,0.0000
P00061=1.575,-3.405,-0.752,0.0000,0.0000,0.0000
P00062=-0.135,-0.848,-1.706,0.0000,0.0000,0.0000
P00063=0.036,-0.654,-3.005,0.0000,0.0000,0.0000
P00100=1.890,0.539,-2.641,0.0000,0.0000,0.0000
//INST
///DATE 2025/02/07 18:49
///ATTR SC,RW
///GROUP1 RB1,BS1
///GROUP2 ST1
NOP
'MUZYLO 300124
'MUZYLO 310124
'POPRAWA I SPAWANIE
'OK_R2_o55a(90,180)
'Path S3739
SFTOF3D
CALL JOB:CLEAN-R1_KM_NEW
MOVJ C00000 BC00000 VJ=100.00  +MOVJ EC00000 VJ=100.00
MOVL C00001 BC00001 V=133.3  +MOVJ EC00001 VJ=100.00
SMOVL C00002 BC00002 V=83.3  +MOVJ EC00002
SREFP 3 C00003 BC00003  +REFP EC00003
CALL JOB:SEARCH-R1-S13D
SET P021 P006
SFTON3D P021
SMOVL C00004 BC00004 V=83.3  +MOVJ EC00004
SREFP 3 C00005 BC00005  +REFP EC00005
CALL JOB:SEARCH-R1-S13D
SET P021 P006
SFTON3D P021
SMOVL C00006 BC00006 V=83.3  +MOVJ EC00006
SREFP 3 C00007 BC00007  +REFP EC00007
CALL JOB:SEARCH-R1-S13D
SET P021 P006
SFTON3D P021
SMOVL C00008 BC00008 V=83.3  +MOVJ EC00008
MOVL C00009 BC00009 V=166.7  +MOVJ EC00009 VJ=100.00
MOVL C00010 BC00010 V=250.0  +MOVJ EC00010 VJ=100.00
'Path S3740
SFTOF3D
MOVJ C00011 BC00011 VJ=100.00  +MOVJ EC00011 VJ=100.00
MOVL C00012 BC00012 V=250.0  +MOVJ EC00012 VJ=100.00
SMOVL C00013 BC00013 V=83.3  +MOVJ EC00013
SREFP 3 C00014 BC00014  +REFP EC00014
CALL JOB:SEARCH-R1-S13D
SET P022 P006
SFTON3D P022
SMOVL C00015 BC00015 V=83.3  +MOVJ EC00015
SREFP 3 C00016 BC00016  +REFP EC00016
CALL JOB:SEARCH-R1-S13D
SET P022 P006
SFTON3D P022
SMOVL C00017 BC00017 V=83.3  +MOVJ EC00017
MOVL C00018 BC00018 V=250.0  +MOVJ EC00018 VJ=100.00
MOVL C00019 BC00019 V=250.0  +MOVJ EC00019 VJ=100.00
MOVJ C00020 BC00020 VJ=100.00  +MOVJ EC00020 VJ=100.00
'
'Path S3741
SFTOF3D
MOVJ C00021 BC00021 VJ=100.00  +MOVJ EC00021 VJ=100.00
MOVL C00022 BC00022 V=250.0  +MOVJ EC00022 VJ=100.00
SMOVL C00023 BC00023 V=83.3  +MOVJ EC00023
SREFP 3 C00024 BC00024  +REFP EC00024
CALL JOB:SEARCH-R1-S13D
SET P031 P006
SFTON3D P031
SMOVL C00025 BC00025 V=83.3  +MOVJ EC00025
SREFP 3 C00026 BC00026  +REFP EC00026
CALL JOB:SEARCH-R1-S13D
SET P031 P006
SFTON3D P031
SMOVL C00027 BC00027 V=83.3  +MOVJ EC00027
SREFP 3 C00028 BC00028  +REFP EC00028
CALL JOB:SEARCH-R1-S13D
SET P031 P006
SFTON3D P031
SMOVL C00029 BC00029 V=83.3  +MOVJ EC00029
MOVL C00030 BC00030 V=166.7  +MOVJ EC00030 VJ=100.00
MOVL C00031 BC00031 V=250.0  +MOVJ EC00031 VJ=100.00
'Path S3742
SFTOF3D
MOVJ C00032 BC00032 VJ=100.00  +MOVJ EC00032 VJ=100.00
MOVL C00033 BC00033 V=333.3  +MOVJ EC00033 VJ=100.00
SMOVL C00034 BC00034 V=83.3  +MOVJ EC00034
SREFP 3 C00035 BC00035  +REFP EC00035
CALL JOB:SEARCH-R1-S13D
SET P032 P006
SFTON3D P032
SMOVL C00036 BC00036 V=83.3  +MOVJ EC00036
SREFP 3 C00037 BC00037  +REFP EC00037
CALL JOB:SEARCH-R1-S13D
SET P032 P006
SFTON3D P032
SMOVL C00038 BC00038 V=83.3  +MOVJ EC00038
MOVL C00039 BC00039 V=166.7  +MOVJ EC00039 VJ=100.00
MOVL C00040 BC00040 V=333.3  +MOVJ EC00040 VJ=100.00
MOVJ C00041 BC00041 VJ=100.00  +MOVJ EC00041 VJ=100.00
'
'Path S3743
SFTOF3D
MOVJ C00042 BC00042 VJ=100.00  +MOVJ EC00042 VJ=100.00
MOVL C00043 BC00043 V=166.7  +MOVJ EC00043 VJ=100.00
SMOVL C00044 BC00044 V=83.3  +MOVJ EC00044
SREFP 3 C00045 BC00045  +REFP EC00045
CALL JOB:SEARCH-R1-S13D
SET P041 P006
SFTON3D P041
SMOVL C00046 BC00046 V=83.3  +MOVJ EC00046
SREFP 3 C00047 BC00047  +REFP EC00047
CALL JOB:SEARCH-R1-S13D
SET P041 P006
SFTON3D P041
SMOVL C00048 BC00048 V=83.3  +MOVJ EC00048
SREFP 3 C00049 BC00049  +REFP EC00049
CALL JOB:SEARCH-R1-S13D
SET P041 P006
SFTON3D P041
SMOVL C00050 BC00050 V=83.3  +MOVJ EC00050
MOVL C00051 BC00051 V=166.7  +MOVJ EC00051 VJ=100.00
MOVL C00052 BC00052 V=250.0  +MOVJ EC00052 VJ=100.00
'Path S3744
SFTOF3D
MOVJ C00053 BC00053 VJ=100.00  +MOVJ EC00053 VJ=100.00
MOVL C00054 BC00054 V=166.7  +MOVJ EC00054 VJ=100.00
SMOVL C00055 BC00055 V=83.3  +MOVJ EC00055
SREFP 3 C00056 BC00056  +REFP EC00056
CALL JOB:SEARCH-R1-S13D
SET P042 P006
SFTON3D P042
SMOVL C00057 BC00057 V=83.3  +MOVJ EC00057
SREFP 3 C00058 BC00058  +REFP EC00058
CALL JOB:SEARCH-R1-S13D
SET P042 P006
SFTON3D P042
SMOVL C00059 BC00059 V=83.3  +MOVJ EC00059
MOVL C00060 BC00060 V=250.0  +MOVJ EC00060 VJ=100.00
MOVL C00061 BC00061 V=333.3  +MOVJ EC00061 VJ=100.00
MOVJ C00062 BC00062 VJ=100.00  +MOVJ EC00062 VJ=100.00
'
'Path S3745
SFTOF3D
MOVJ C00063 BC00063 VJ=100.00  +MOVJ EC00063 VJ=100.00
MOVL C00064 BC00064 V=166.7  +MOVJ EC00064 VJ=100.00
SMOVL C00065 BC00065 V=83.3  +MOVJ EC00065
SREFP 3 C00066 BC00066  +REFP EC00066
CALL JOB:SEARCH-R1-S13D
SET P051 P006
SFTON3D P051
SMOVL C00067 BC00067 V=83.3  +MOVJ EC00067
SREFP 3 C00068 BC00068  +REFP EC00068
CALL JOB:SEARCH-R1-S13D
SET P051 P006
SFTON3D P051
SMOVL C00069 BC00069 V=83.3  +MOVJ EC00069
SREFP 3 C00070 BC00070  +REFP EC00070
CALL JOB:SEARCH-R1-S13D
SET P051 P006
SFTON3D P051
SMOVL C00071 BC00071 V=83.3  +MOVJ EC00071
MOVL C00072 BC00072 V=166.7  +MOVJ EC00072 VJ=100.00
MOVL C00073 BC00073 V=250.0  +MOVJ EC00073 VJ=100.00
'Path S3746
SFTOF3D
MOVJ C00074 BC00074 VJ=100.00  +MOVJ EC00074 VJ=100.00
MOVL C00075 BC00075 V=166.7  +MOVJ EC00075 VJ=100.00
SMOVL C00076 BC00076 V=83.3  +MOVJ EC00076
SREFP 3 C00077 BC00077  +REFP EC00077
CALL JOB:SEARCH-R1-S13D
SET P052 P006
SFTON3D P052
SMOVL C00078 BC00078 V=83.3  +MOVJ EC00078
SREFP 3 C00079 BC00079  +REFP EC00079
CALL JOB:SEARCH-R1-S13D
SET P052 P006
SFTON3D P052
SMOVL C00080 BC00080 V=83.3  +MOVJ EC00080
MOVL C00081 BC00081 V=166.7  +MOVJ EC00081 VJ=100.00
MOVL C00082 BC00082 V=250.0  +MOVJ EC00082 VJ=100.00
MOVJ C00083 BC00083 VJ=100.00  +MOVJ EC00083 VJ=100.00
'
'Path S3747
SFTOF3D
MOVJ C00084 BC00084 VJ=100.00  +MOVJ EC00084 VJ=100.00
MOVL C00085 BC00085 V=250.0  +MOVJ EC00085 VJ=100.00
SMOVL C00086 BC00086 V=83.3  +MOVJ EC00086
SREFP 3 C00087 BC00087  +REFP EC00087
CALL JOB:SEARCH-R1-S13D
SET P061 P006
SFTON3D P061
SMOVL C00088 BC00088 V=83.3  +MOVJ EC00088
SREFP 3 C00089 BC00089  +REFP EC00089
CALL JOB:SEARCH-R1-S13D
SET P061 P006
SFTON3D P061
SMOVL C00090 BC00090 V=83.3  +MOVJ EC00090
SREFP 3 C00091 BC00091  +REFP EC00091
CALL JOB:SEARCH-R1-S13D
SET P061 P006
SFTON3D P061
SMOVL C00092 BC00092 V=83.3  +MOVJ EC00092
MOVL C00093 BC00093 V=166.7  +MOVJ EC00093 VJ=100.00
MOVL C00094 BC00094 V=250.0  +MOVJ EC00094 VJ=100.00
'Path S3748
SFTOF3D
MOVJ C00095 BC00095 VJ=100.00  +MOVJ EC00095 VJ=100.00
MOVL C00096 BC00096 V=166.7  +MOVJ EC00096 VJ=100.00
SMOVL C00097 BC00097 V=83.3  +MOVJ EC00097
SREFP 3 C00098 BC00098  +REFP EC00098
CALL JOB:SEARCH-R1-S13D
SET P062 P006
SFTON3D P062
SMOVL C00099 BC00099 V=83.3  +MOVJ EC00099
SREFP 3 C00100 BC00100  +REFP EC00100
CALL JOB:SEARCH-R1-S13D
SET P062 P006
SFTON3D P062
SMOVL C00101 BC00101 V=83.3  +MOVJ EC00101
MOVL C00102 BC00102 V=166.7  +MOVJ EC00102 VJ=100.00
MOVL C00103 BC00103 V=250.0  +MOVJ EC00103 VJ=100.00
MOVJ C00104 BC00104 VJ=100.00  +MOVJ EC00104 VJ=100.00
'
MOVJ C00105 BC00105 VJ=100.00  +MOVJ EC00105 VJ=100.00
MOVJ C00106 BC00106 VJ=100.00  +MOVJ EC00106 VJ=100.00
SFTOF3D
MOVJ C00107 BC00107 VJ=100.00  +MOVJ EC00107 VJ=100.00
SMOVL C00108 BC00108 V=83.3  +MOVJ EC00108
SREFP 3 C00109 BC00109  +REFP EC00109
CALL JOB:SEARCH-R1-S13D
SET P100 P006
SFTON3D P100
SMOVL C00110 BC00110 V=83.3  +MOVJ EC00110
SMOVL C00111 BC00111 V=133.3  +MOVJ EC00111
SMOVL C00112 BC00112 V=83.3  +MOVJ EC00112
SREFP 3 C00113 BC00113  +REFP EC00113
CALL JOB:SEARCH-R1-S13D
SET P100 P006
SFTON3D P100
SMOVL C00114 BC00114 V=83.3  +MOVJ EC00114
SMOVL C00115 BC00115 V=166.7  +MOVJ EC00115
SREFP 3 C00116 BC00116  +REFP EC00116
CALL JOB:SEARCH-R1-S13D
SET P100 P006
SFTON3D P100
SMOVL C00117 BC00117 V=166.7  +MOVJ EC00117
SMOVL C00118 BC00118 V=166.7  +MOVJ EC00118
MOVJ C00119 BC00119 VJ=100.00  +MOVJ EC00119 VJ=100.00
'Path S3749
SFTOF3D
MOVJ C00120 BC00120 VJ=100.00  +MOVJ EC00120 VJ=100.00
MOVL C00121 BC00121 V=166.7  +MOVJ EC00121 VJ=100.00
SMOVL C00122 BC00122 V=83.3  +MOVJ EC00122
SREFP 3 C00123 BC00123  +REFP EC00123
CALL JOB:SEARCH-R1-S13D
SET P063 P006
SFTON3D P063
SMOVL C00124 BC00124 V=83.3  +MOVJ EC00124
SREFP 3 C00125 BC00125  +REFP EC00125
CALL JOB:SEARCH-R1-S13D
SET P063 P006
SFTON3D P063
SMOVL C00126 BC00126 V=83.3  +MOVJ EC00126
MOVL C00127 BC00127 V=166.7  +MOVJ EC00127 VJ=100.00
MOVL C00128 BC00128 V=250.0  +MOVJ EC00128 VJ=100.00
'Path S3750
SFTOF3D
MOVJ C00129 BC00129 VJ=100.00  +MOVJ EC00129 VJ=100.00
MOVL C00130 BC00130 V=250.0  +MOVJ EC00130 VJ=100.00
SMOVL C00131 BC00131 V=83.3  +MOVJ EC00131
SREFP 3 C00132 BC00132  +REFP EC00132
CALL JOB:SEARCH-R1-S13D
SET P053 P006
SFTON3D P053
SMOVL C00133 BC00133 V=83.3  +MOVJ EC00133
SREFP 3 C00134 BC00134  +REFP EC00134
CALL JOB:SEARCH-R1-S13D
SET P053 P006
SFTON3D P053
SMOVL C00135 BC00135 V=83.3  +MOVJ EC00135
MOVL C00136 BC00136 V=166.7  +MOVJ EC00136 VJ=100.00
MOVL C00137 BC00137 V=250.0  +MOVJ EC00137 VJ=100.00
'Path S3751
SFTOF3D
MOVJ C00138 BC00138 VJ=100.00  +MOVJ EC00138 VJ=100.00
MOVL C00139 BC00139 V=250.0  +MOVJ EC00139 VJ=100.00
SMOVL C00140 BC00140 V=83.3  +MOVJ EC00140
SREFP 3 C00141 BC00141  +REFP EC00141
CALL JOB:SEARCH-R1-S13D
SET P043 P006
SFTON3D P043
SMOVL C00142 BC00142 V=83.3  +MOVJ EC00142
SREFP 3 C00143 BC00143  +REFP EC00143
CALL JOB:SEARCH-R1-S13D
SET P043 P006
SFTON3D P043
SMOVL C00144 BC00144 V=83.3  +MOVJ EC00144
MOVL C00145 BC00145 V=166.7  +MOVJ EC00145 VJ=100.00
MOVL C00146 BC00146 V=250.0  +MOVJ EC00146 VJ=100.00
'Path S3752
SFTOF3D
MOVJ C00147 BC00147 VJ=100.00  +MOVJ EC00147 VJ=100.00
MOVL C00148 BC00148 V=166.7  +MOVJ EC00148 VJ=100.00
SMOVL C00149 BC00149 V=83.3  +MOVJ EC00149
SREFP 3 C00150 BC00150  +REFP EC00150
CALL JOB:SEARCH-R1-S13D
SET P033 P006
SFTON3D P033
SMOVL C00151 BC00151 V=83.3  +MOVJ EC00151
SREFP 3 C00152 BC00152  +REFP EC00152
CALL JOB:SEARCH-R1-S13D
SET P033 P006
SFTON3D P033
SMOVL C00153 BC00153 V=83.3  +MOVJ EC00153
MOVL C00154 BC00154 V=166.7  +MOVJ EC00154 VJ=100.00
MOVL C00155 BC00155 V=250.0  +MOVJ EC00155 VJ=100.00
'Path S3753
SFTOF3D
MOVJ C00156 BC00156 VJ=100.00  +MOVJ EC00156 VJ=100.00
MOVL C00157 BC00157 V=250.0  +MOVJ EC00157 VJ=100.00
SMOVL C00158 BC00158 V=83.3  +MOVJ EC00158
SREFP 3 C00159 BC00159  +REFP EC00159
CALL JOB:SEARCH-R1-S13D
SET P023 P006
SFTON3D P023
SMOVL C00160 BC00160 V=83.3  +MOVJ EC00160
SREFP 3 C00161 BC00161  +REFP EC00161
CALL JOB:SEARCH-R1-S13D
SET P023 P006
SFTON3D P023
SMOVL C00162 BC00162 V=83.3  +MOVJ EC00162
MOVL C00163 BC00163 V=166.7  +MOVJ EC00163 VJ=100.00
MOVL C00164 BC00164 V=250.0  +MOVJ EC00164 VJ=100.00
'
'
'
'Path W3754
SFTOF3D
SFTON3D P043
MOVJ C00165 BC00165 VJ=100.00  +MOVJ EC00165 VJ=100.00
SMOVL C00166 BC00166 V=166.7  +MOVJ EC00166
SMOVL C00167 BC00167 V=133.3 PL=0  +MOVJ EC00167
SREFP 1 C00168 BC00168  +REFP EC00168
SREFP 2 C00169 BC00169  +REFP EC00169
MACRO1 MJ#(0) ARGF9
ARCON
SMOVL C00170 BC00170 V=9.2  +MOVJ EC00170
SMOVL C00171 BC00171 V=9.2  +MOVJ EC00171
SMOVL C00172 BC00172 V=9.2  +MOVJ EC00172
ARCOF
SMOVL C00173 BC00173 V=133.3  +MOVJ EC00173
SMOVL C00174 BC00174 V=250.0  +MOVJ EC00174
SFTOF3D
'Path W3755
SFTOF3D
SFTON3D P023
MOVJ C00175 BC00175 VJ=100.00  +MOVJ EC00175 VJ=100.00
SMOVL C00176 BC00176 V=250.0  +MOVJ EC00176
SMOVL C00177 BC00177 V=133.3 PL=0  +MOVJ EC00177
SREFP 1 C00178 BC00178  +REFP EC00178
SREFP 2 C00179 BC00179  +REFP EC00179
ARCON
SMOVL C00180 BC00180 V=9.2  +MOVJ EC00180
SMOVL C00181 BC00181 V=9.2  +MOVJ EC00181
SMOVL C00182 BC00182 V=9.2  +MOVJ EC00182
ARCOF
SMOVL C00183 BC00183 V=133.3  +MOVJ EC00183
SMOVL C00184 BC00184 V=250.0  +MOVJ EC00184
SFTOF3D
'Path W3756
SFTOF3D
SFTON3D P063
MOVJ C00185 BC00185 VJ=100.00  +MOVJ EC00185 VJ=100.00
SMOVL C00186 BC00186 V=166.7  +MOVJ EC00186
SMOVL C00187 BC00187 V=166.7 PL=0  +MOVJ EC00187
SREFP 1 C00188 BC00188  +REFP EC00188
SREFP 2 C00189 BC00189  +REFP EC00189
MACRO1 MJ#(0) ARGF9
ARCON
SMOVL C00190 BC00190 V=9.2  +MOVJ EC00190
SMOVL C00191 BC00191 V=9.2  +MOVJ EC00191
SMOVL C00192 BC00192 V=9.2  +MOVJ EC00192
SMOVL C00193 BC00193 V=9.2  +MOVJ EC00193
ARCOF
SMOVL C00194 BC00194 V=250.0  +MOVJ EC00194
SMOVL C00195 BC00195 V=666.7  +MOVJ EC00195
SFTOF3D
'Path W3757
SFTOF3D
SFTON3D P033
MOVJ C00196 BC00196 VJ=100.00  +MOVJ EC00196 VJ=100.00
SMOVL C00197 BC00197 V=500.0  +MOVJ EC00197
SMOVL C00198 BC00198 V=200.0 PL=0  +MOVJ EC00198
SREFP 1 C00199 BC00199  +REFP EC00199
SREFP 2 C00200 BC00200  +REFP EC00200
ARCON
SMOVL C00201 BC00201 V=9.2  +MOVJ EC00201
SMOVL C00202 BC00202 V=9.2  +MOVJ EC00202
SMOVL C00203 BC00203 V=9.2  +MOVJ EC00203
SMOVL C00204 BC00204 V=9.2  +MOVJ EC00204
ARCOF
SMOVL C00205 BC00205 V=250.0  +MOVJ EC00205
SMOVL C00206 BC00206 V=500.0  +MOVJ EC00206
SFTOF3D
'Path W3758
SFTOF3D
SFTON3D P053
MOVJ C00207 BC00207 VJ=100.00  +MOVJ EC00207 VJ=100.00
SMOVL C00208 BC00208 V=500.0  +MOVJ EC00208
SMOVL C00209 BC00209 V=250.0 PL=0  +MOVJ EC00209
SREFP 1 C00210 BC00210  +REFP EC00210
SREFP 2 C00211 BC00211  +REFP EC00211
ARCON
SMOVL C00212 BC00212 V=9.2  +MOVJ EC00212
SMOVL C00213 BC00213 V=9.2  +MOVJ EC00213
SMOVL C00214 BC00214 V=9.2  +MOVJ EC00214
SMOVL C00215 BC00215 V=9.2  +MOVJ EC00215
ARCOF
SMOVL C00216 BC00216 V=250.0  +MOVJ EC00216
SMOVL C00217 BC00217 V=666.7  +MOVJ EC00217
SFTOF3D
MOVJ C00218 BC00218 VJ=100.00  +MOVJ EC00218 VJ=100.00
MOVJ C00219 BC00219 VJ=100.00  +MOVJ EC00219 VJ=100.00
'
MOVJ C00220 BC00220 VJ=100.00  +MOVJ EC00220 VJ=100.00
SFTOF3D
SFTON3D P042
MOVJ C00221 BC00221 VJ=100.00  +MOVJ EC00221 VJ=100.00
SMOVL C00222 BC00222 V=166.7  +MOVJ EC00222
SMOVL C00223 BC00223 V=250.0 PL=0  +MOVJ EC00223
SREFP 1 C00224 BC00224  +REFP EC00224
SREFP 2 C00225 BC00225  +REFP EC00225
ARCON
SMOVL C00226 BC00226 V=9.2  +MOVJ EC00226
SMOVL C00227 BC00227 V=9.2  +MOVJ EC00227
SMOVL C00228 BC00228 V=9.2  +MOVJ EC00228
SMOVL C00229 BC00229 V=9.2  +MOVJ EC00229
SMOVL C00230 BC00230 V=9.2  +MOVJ EC00230
SFTON3D P041
SMOVL C00231 BC00231 V=9.2  +MOVJ EC00231
SMOVL C00232 BC00232 V=9.2  +MOVJ EC00232
ARCOF
SMOVL C00233 BC00233 V=250.0  +MOVJ EC00233
SMOVL C00234 BC00234 V=666.7  +MOVJ EC00234
SFTOF3D
'Path W3761
SFTOF3D
SFTON3D P041
MOVJ C00235 BC00235 VJ=100.00  +MOVJ EC00235 VJ=100.00
SMOVL C00236 BC00236 V=666.7  +MOVJ EC00236
SMOVL C00237 BC00237 V=250.0 PL=0  +MOVJ EC00237
SREFP 1 C00238 BC00238  +REFP EC00238
SREFP 2 C00239 BC00239  +REFP EC00239
ARCON
SMOVL C00240 BC00240 V=9.2  +MOVJ EC00240
SMOVL C00241 BC00241 V=9.2  +MOVJ EC00241
ARCOF
SMOVL C00242 BC00242 V=250.0  +MOVJ EC00242
SMOVL C00243 BC00243 V=666.7  +MOVJ EC00243
SFTOF3D
MOVJ C00244 BC00244 VJ=100.00  +MOVJ EC00244 VJ=100.00
'
'
MOVJ C00245 BC00245 VJ=100.00  +MOVJ EC00245 VJ=100.00
'Path W3762
SFTOF3D
SFTON3D P022
MOVJ C00246 BC00246 VJ=100.00  +MOVJ EC00246 VJ=100.00
SMOVL C00247 BC00247 V=166.7  +MOVJ EC00247
SMOVL C00248 BC00248 V=250.0 PL=0  +MOVJ EC00248
SREFP 1 C00249 BC00249  +REFP EC00249
SREFP 2 C00250 BC00250  +REFP EC00250
ARCON
SMOVL C00251 BC00251 V=9.2  +MOVJ EC00251
SMOVL C00252 BC00252 V=9.2  +MOVJ EC00252
ARCOF
SMOVL C00253 BC00253 V=250.0  +MOVJ EC00253
SMOVL C00254 BC00254 V=666.7  +MOVJ EC00254
SFTOF3D
'Path W3763
SFTOF3D
SFTON3D P021
MOVJ C00255 BC00255 VJ=100.00  +MOVJ EC00255 VJ=100.00
SMOVL C00256 BC00256 V=166.7  +MOVJ EC00256
SMOVL C00257 BC00257 V=250.0 PL=0  +MOVJ EC00257
SREFP 1 C00258 BC00258  +REFP EC00258
SREFP 2 C00259 BC00259  +REFP EC00259
ARCON
SMOVL C00260 BC00260 V=9.2  +MOVJ EC00260
SMOVL C00261 BC00261 V=9.2  +MOVJ EC00261
SMOVL C00262 BC00262 V=9.2  +MOVJ EC00262
ARCOF
SMOVL C00263 BC00263 V=250.0  +MOVJ EC00263
SMOVL C00264 BC00264 V=666.7  +MOVJ EC00264
SFTOF3D
'Path W3764
SFTOF3D
SFTON3D P021
MOVJ C00265 BC00265 VJ=100.00  +MOVJ EC00265 VJ=100.00
SMOVL C00266 BC00266 V=666.7  +MOVJ EC00266
SMOVL C00267 BC00267 V=250.0 PL=0  +MOVJ EC00267
SREFP 1 C00268 BC00268  +REFP EC00268
SREFP 2 C00269 BC00269  +REFP EC00269
ARCON
SMOVL C00270 BC00270 V=9.2  +MOVJ EC00270
SMOVL C00271 BC00271 V=9.2  +MOVJ EC00271
SMOVL C00272 BC00272 V=9.2  +MOVJ EC00272
ARCOF
SMOVL C00273 BC00273 V=250.0  +MOVJ EC00273
SMOVL C00274 BC00274 V=666.7  +MOVJ EC00274
SFTOF3D
MOVJ C00275 BC00275 VJ=100.00  +MOVJ EC00275 VJ=100.00
'
'
MOVJ C00276 BC00276 VJ=100.00  +MOVJ EC00276 VJ=100.00
'Path W3765
SFTOF3D
SFTON3D P062
MOVJ C00277 BC00277 VJ=100.00  +MOVJ EC00277 VJ=100.00
SMOVL C00278 BC00278 V=666.7  +MOVJ EC00278
SMOVL C00279 BC00279 V=250.0 PL=0  +MOVJ EC00279
SREFP 1 C00280 BC00280  +REFP EC00280
SREFP 2 C00281 BC00281  +REFP EC00281
ARCON
SMOVL C00282 BC00282 V=9.2  +MOVJ EC00282
SMOVL C00283 BC00283 V=9.2  +MOVJ EC00283
ARCOF
SMOVL C00284 BC00284 V=250.0  +MOVJ EC00284
SMOVL C00285 BC00285 V=666.7  +MOVJ EC00285
SFTOF3D
'Path W3766
SFTOF3D
SFTON3D P061
MOVJ C00286 BC00286 VJ=100.00  +MOVJ EC00286 VJ=100.00
SMOVL C00287 BC00287 V=666.7  +MOVJ EC00287
SMOVL C00288 BC00288 V=250.0 PL=0  +MOVJ EC00288
SREFP 1 C00289 BC00289  +REFP EC00289
SREFP 2 C00290 BC00290  +REFP EC00290
ARCON
SMOVL C00291 BC00291 V=9.2  +MOVJ EC00291
SMOVL C00292 BC00292 V=9.2  +MOVJ EC00292
SMOVL C00293 BC00293 V=9.2  +MOVJ EC00293
ARCOF
SMOVL C00294 BC00294 V=250.0  +MOVJ EC00294
SMOVL C00295 BC00295 V=666.7  +MOVJ EC00295
SFTOF3D
'Path W3767
SFTOF3D
SFTON3D P061
MOVJ C00296 BC00296 VJ=100.00  +MOVJ EC00296 VJ=100.00
SMOVL C00297 BC00297 V=666.7  +MOVJ EC00297
SMOVL C00298 BC00298 V=250.0 PL=0  +MOVJ EC00298
SREFP 1 C00299 BC00299  +REFP EC00299
SREFP 2 C00300 BC00300  +REFP EC00300
ARCON
SMOVL C00301 BC00301 V=9.2  +MOVJ EC00301
SMOVL C00302 BC00302 V=9.2  +MOVJ EC00302
ARCOF
SMOVL C00303 BC00303 V=250.0  +MOVJ EC00303
SMOVL C00304 BC00304 V=666.7  +MOVJ EC00304
SFTOF3D
MOVJ C00305 BC00305 VJ=100.00  +MOVJ EC00305 VJ=100.00
'
'
MOVJ C00306 BC00306 VJ=100.00  +MOVJ EC00306 VJ=100.00
'Path W3768
SFTOF3D
SFTON3D P032
MOVJ C00307 BC00307 VJ=100.00  +MOVJ EC00307 VJ=100.00
SMOVL C00308 BC00308 V=666.7  +MOVJ EC00308
SMOVL C00309 BC00309 V=250.0 PL=0  +MOVJ EC00309
SREFP 1 C00310 BC00310  +REFP EC00310
SREFP 2 C00311 BC00311  +REFP EC00311
ARCON
SMOVL C00312 BC00312 V=9.2  +MOVJ EC00312
SMOVL C00313 BC00313 V=9.2  +MOVJ EC00313
ARCOF
SMOVL C00314 BC00314 V=250.0  +MOVJ EC00314
SMOVL C00315 BC00315 V=666.7  +MOVJ EC00315
SFTOF3D
'Path W3769
SFTOF3D
SFTON3D P031
MOVJ C00316 BC00316 VJ=100.00  +MOVJ EC00316 VJ=100.00
SMOVL C00317 BC00317 V=666.7  +MOVJ EC00317
SMOVL C00318 BC00318 V=250.0 PL=0  +MOVJ EC00318
SREFP 1 C00319 BC00319  +REFP EC00319
SREFP 2 C00320 BC00320  +REFP EC00320
ARCON
SMOVL C00321 BC00321 V=9.2  +MOVJ EC00321
SMOVL C00322 BC00322 V=9.2  +MOVJ EC00322
SMOVL C00323 BC00323 V=9.2  +MOVJ EC00323
SMOVL C00324 BC00324 V=9.2  +MOVJ EC00324
ARCOF
SMOVL C00325 BC00325 V=250.0  +MOVJ EC00325
SMOVL C00326 BC00326 V=666.7  +MOVJ EC00326
SFTOF3D
'Path W3770
SFTOF3D
SFTON3D P031
MOVJ C00327 BC00327 VJ=100.00  +MOVJ EC00327 VJ=100.00
SMOVL C00328 BC00328 V=666.7  +MOVJ EC00328
SMOVL C00329 BC00329 V=200.0 PL=0  +MOVJ EC00329
SREFP 1 C00330 BC00330  +REFP EC00330
SREFP 2 C00331 BC00331  +REFP EC00331
ARCON
SMOVL C00332 BC00332 V=9.2  +MOVJ EC00332
SMOVL C00333 BC00333 V=9.2  +MOVJ EC00333
SMOVL C00334 BC00334 V=9.2  +MOVJ EC00334
ARCOF
SMOVL C00335 BC00335 V=200.0  +MOVJ EC00335
SMOVL C00336 BC00336 V=666.7  +MOVJ EC00336
SFTOF3D
MOVJ C00337 BC00337 VJ=100.00  +MOVJ EC00337 VJ=100.00
'
'
MOVJ C00338 BC00338 VJ=100.00  +MOVJ EC00338 VJ=100.00
'Path W3771
SFTOF3D
SFTON3D P052
MOVJ C00339 BC00339 VJ=100.00  +MOVJ EC00339 VJ=100.00
SMOVL C00340 BC00340 V=666.7  +MOVJ EC00340
SMOVL C00341 BC00341 V=200.0 PL=0  +MOVJ EC00341
SREFP 1 C00342 BC00342  +REFP EC00342
SREFP 2 C00343 BC00343  +REFP EC00343
ARCON
SMOVL C00344 BC00344 V=9.2  +MOVJ EC00344
SMOVL C00345 BC00345 V=9.2  +MOVJ EC00345
ARCOF
SMOVL C00346 BC00346 V=133.3  +MOVJ EC00346
SMOVL C00347 BC00347 V=250.0  +MOVJ EC00347
SFTOF3D
'Path W3772
SFTOF3D
SFTON3D P051
MOVJ C00348 BC00348 VJ=100.00  +MOVJ EC00348 VJ=100.00
SMOVL C00349 BC00349 V=666.7  +MOVJ EC00349
SMOVL C00350 BC00350 V=200.0 PL=0  +MOVJ EC00350
ARCON
SREFP 1 C00351 BC00351  +REFP EC00351
SREFP 2 C00352 BC00352  +REFP EC00352
SMOVL C00353 BC00353 V=9.2  +MOVJ EC00353
SMOVL C00354 BC00354 V=9.2  +MOVJ EC00354
SMOVL C00355 BC00355 V=9.2  +MOVJ EC00355
SMOVL C00356 BC00356 V=9.2  +MOVJ EC00356
ARCOF
SMOVL C00357 BC00357 V=250.0  +MOVJ EC00357
SMOVL C00358 BC00358 V=666.7  +MOVJ EC00358
SFTOF3D
'Path W3773
SFTOF3D
SFTON3D P051
MOVJ C00359 BC00359 VJ=100.00  +MOVJ EC00359 VJ=100.00
SMOVL C00360 BC00360 V=666.7  +MOVJ EC00360
SMOVL C00361 BC00361 V=200.0 PL=0  +MOVJ EC00361
SREFP 1 C00362 BC00362  +REFP EC00362
SREFP 2 C00363 BC00363  +REFP EC00363
ARCON
SMOVL C00364 BC00364 V=9.2  +MOVJ EC00364
SMOVL C00365 BC00365 V=9.2  +MOVJ EC00365
SMOVL C00366 BC00366 V=9.2  +MOVJ EC00366
ARCOF
SMOVL C00367 BC00367 V=250.0  +MOVJ EC00367
SMOVL C00368 BC00368 V=666.7  +MOVJ EC00368
SFTOF3D
MOVJ C00369 BC00369 VJ=100.00  +MOVJ EC00369 VJ=100.00
MOVJ C00370 BC00370 VJ=100.00  +MOVJ EC00370 VJ=100.00
SFTOF3D
MOVJ C00371 BC00371 VJ=100.00  +MOVJ EC00371 VJ=100.00
SFTON3D P100
SMOVL C00372 BC00372 V=166.7 PL=0  +MOVJ EC00372
ARCON
SWVON WEV#(102)
SMOVL C00373 BC00373 V=8.3  +MOVJ EC00373
SMOVL C00374 BC00374 V=8.3  +MOVJ EC00374
ARCOF
SWVOF
SMOVL C00375 BC00375 V=250.0  +MOVJ EC00375
MACRO1 MJ#(0) ARGF14
SMOVL C00376 BC00376 V=666.7  +MOVJ EC00376
SMOVL C00377 BC00377 V=200.0 PL=0  +MOVJ EC00377
ARCON
SWVON WEV#(66)
SMOVL C00378 BC00378 V=10.8  +MOVJ EC00378
SMOVL C00379 BC00379 V=10.8  +MOVJ EC00379
ARCON
SMOVL C00380 BC00380 V=10.8  +MOVJ EC00380
SMOVL C00381 BC00381 V=10.8  +MOVJ EC00381
SMOVL C00382 BC00382 V=10.8  +MOVJ EC00382
SMOVL C00383 BC00383 V=10.8  +MOVJ EC00383
ARCOF
SWVOF
SFTOF3D
SMOVL C00384 BC00384 V=250.0  +MOVJ EC00384
MOVJ C00385 BC00385 VJ=100.00  +MOVJ EC00385 VJ=100.00
'
END
